INTERFACE I_XtsTrack

PROPERTY IsTrackSetForDetection : BOOL
GET
END_GET
END_PROPERTY

PROPERTY MyOTCID : OTCID
GET
END_GET
SET
END_SET
END_PROPERTY

METHOD RemoveFromDetection : BOOL
VAR_INPUT
END_VAR
END_METHOD

METHOD SetForDetection : BOOL
VAR_INPUT
END_VAR
END_METHOD

PROPERTY TrackLength : MC_Lreal
GET
END_GET
END_PROPERTY

END_INTERFACE

(* stored: Version 1.1.0.1
   Itf I_XtsTrack: Id {b580e084-f2aa-4b9e-b34b-5773df679de5}
   Property IsTrackSetForDetection: Id {b3d46c63-3436-40e6-816c-0d3d6f24401f}
   Get Get: Id {fb5f8c6b-7961-46c2-ac4d-21822b0c9d98}
   Property MyOTCID: Id {8be67bfb-cfe2-4d62-98cc-25000c035505}
   Get Get: Id {4e95c9bb-aa4d-4ade-9bfa-d3c230375802}
   Set Set: Id {5a69d026-ba0e-42f2-ad56-82e6069370de}
   Method RemoveFromDetection: Id {9e7f91cb-3f18-4120-a764-6e1db78d984c}
   Method SetForDetection: Id {025c650b-b106-4b4a-a957-33ebeda4f9a9}
   Property TrackLength: Id {d09b154e-641d-4452-b45a-353375f2a798}
   Get Get: Id {227be027-fd95-4a28-b451-be32068fa3af} *)
